KUKA KRL program: FOLLOWTRIG.src, FOLLOWTRIG.dat

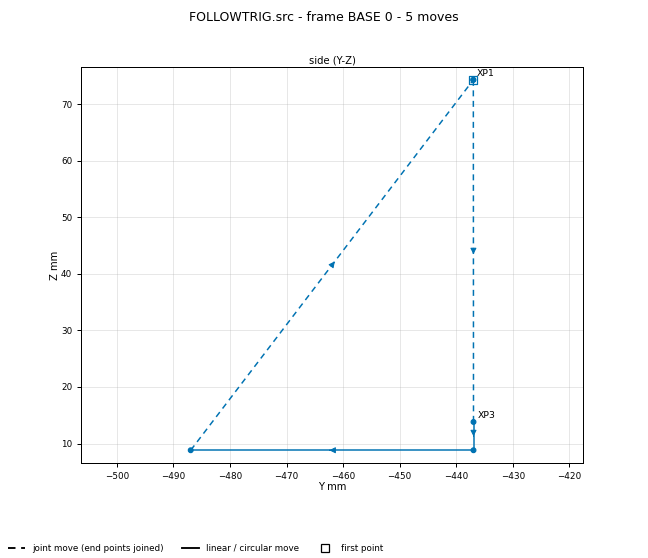
[picture p0: tool path of FOLLOWTRIG.src in frame BASE 0, 5 of 5 moves have a stored position in this frame; points joined in program order, loops and branches not executed]
--- FOLLOWTRIG.src ---
&ACCESS RVO
&REL 127
&PARAM TEMPLATE = C:\KRC\Roboter\Template\vorgabe
&PARAM EDITMASK = *
DEF FOLLOWTRIG( )
DECL TORQUE_TCP_EST MyTorque
DECL BOOL TEMP, HEMP, DEMP
DECL INT TMP1, n, result
DECL INT md_int[16]
DECL REAL md_real[16]
;FOLD INI
  ;FOLD BASISTECH INI
    GLOBAL INTERRUPT DECL 3 WHEN $STOPMESS==TRUE DO IR_STOPM ( )
    INTERRUPT ON 3
    BAS (#INITMOV,0 )
  ;ENDFOLD (BASISTECH INI)
  ;FOLD USER INI
    ;Make your modifications here
  ;ENDFOLD (USER INI)
;ENDFOLD (INI)

$OV_PRO=50
$TOOL=TOOL_DATA[5]
$VEL.CP=1.0
$VEL.ORI1=150
$VEL.ORI2=100
$ACC.CP=1.7
$ACC.ORI1=80
$ACC.ORI2=80
$ORI_TYPE=#CONSTANT

;FOLD PTP P1 Vel=100 % PDAT1 Tool[5]:Pneumatic_gripper_probe Base[0];%{PE}%R 5.6.11,%MKUKATPBASIS,%CMOVE,%VPTP,%P 1:PTP, 2:P1, 3:, 5:100, 7:PDAT1
$BWDSTART=FALSE
PDAT_ACT=PPDAT1
FDAT_ACT=FP1
BAS(#PTP_PARAMS,100)
PTP XP1
;ENDFOLD

;FOLD PTP P3 Vel=100 % PDAT3 Tool[5]:Pneumatic_gripper_probe Base[0];%{PE}%R 5.6.11,%MKUKATPBASIS,%CMOVE,%VPTP,%P 1:PTP, 2:P3, 3:, 5:100, 7:PDAT3
$BWDSTART=FALSE
PDAT_ACT=PPDAT3
FDAT_ACT=FP3
BAS(#PTP_PARAMS,100)
PTP XP3
;ENDFOLD

$STIFFNESS.STRATEGY=10
$STIFFNESS.COMMIT=TRUE
$OV_PRO=25

HALT

HEMP=TRIG()

$OV_PRO=25

LIN_REL {Z -5}

;REPEAT
  ;MyTorque=$TORQUE_TCP_EST
;UNTIL MyTorque.FT.Z >= .1

LIN_REL {Y -50}

HALT

FOR n=1 TO 16
  md_int[n]=0
  md_real[n]=0
ENDFOR

md_real[1]=0.05

result=MD_CMD("PAPAS","TRIGBYCONTACT",md_int[],md_real[])

$STIFFNESS.STRATEGY=10
$STIFFNESS.COMMIT=TRUE
$OV_PRO=25

;FOLD PTP P2 Vel=100 % PDAT2 Tool[5]:Pneumatic_gripper_probe Base[0];%{PE}%R 5.6.11,%MKUKATPBASIS,%CMOVE,%VPTP,%P 1:PTP, 2:P2, 3:, 5:100, 7:PDAT2
$BWDSTART=FALSE
PDAT_ACT=PPDAT2
FDAT_ACT=FP2
BAS(#PTP_PARAMS,100)
PTP XP2
;ENDFOLD

END

--- FOLLOWTRIG.dat ---
&ACCESS RVO
&REL 127
&PARAM TEMPLATE = C:\KRC\Roboter\Template\vorgabe
&PARAM EDITMASK = *
DEFDAT  FOLLOWTRIG
;FOLD EXTERNAL DECLARATIONS;%{PE}%MKUKATPBASIS,%CEXT,%VCOMMON,%P
;FOLD BASISTECH EXT;%{PE}%MKUKATPBASIS,%CEXT,%VEXT,%P
EXT  BAS (BAS_COMMAND  :IN,REAL  :IN )
DECL INT SUCCESS
;ENDFOLD (BASISTECH EXT)
;FOLD USER EXT;%{E}%MKUKATPUSER,%CEXT,%VEXT,%P
;Make here your modifications

;ENDFOLD (USER EXT)
;ENDFOLD (EXTERNAL DECLARATIONS)
DECL BASIS_SUGG_T LAST_BASIS={POINT1[] "P3                      ",POINT2[] "P3                      ",CP_PARAMS[] "CPDAT0                  ",PTP_PARAMS[] "PDAT3                   ",CONT[] "                        ",CP_VEL[] "2.0                     ",PTP_VEL[] "100                     ",SYNC_PARAMS[] "SYNCDAT                 ",SPL_NAME[] "S0                      "}
DECL E6POS XP1={X -559.982727,Y -436.976105,Z 74.2944412,A 89.9887924,B -0.00345713296,C 179.995499,S 1,T 12,E1 0.251655608,E2 0.0,E3 0.0,E4 0.0,E5 0.0,E6 0.0}
DECL FDAT FP1={TOOL_NO 5,BASE_NO 0,IPO_FRAME #BASE,POINT2[] " ",TQ_STATE FALSE}
DECL PDAT PPDAT1={VEL 100.0,ACC 100.0,APO_DIST 100.0,APO_MODE #CPTP}
DECL E6POS XP2={X -559.982422,Y -436.976501,Z 74.2944412,A 89.9887466,B -0.00337572605,C 179.995407,S 1,T 12,E1 0.251655608,E2 0.0,E3 0.0,E4 0.0,E5 0.0,E6 0.0}
DECL FDAT FP2={TOOL_NO 5,BASE_NO 0,IPO_FRAME #BASE,POINT2[] " ",TQ_STATE FALSE}
DECL PDAT PPDAT2={VEL 100.0,ACC 100.0,APO_DIST 100.0,APO_MODE #CPTP}
DECL INT LAST_XP_POINT=2
DECL E6POS XP3={X -559.928772,Y -436.946411,Z 13.8073597,A 89.9849319,B -0.0102660097,C 179.986099,S 1,T 12,E1 0.251947403,E2 0.0,E3 0.0,E4 0.0,E5 0.0,E6 0.0}
DECL FDAT FP3={TOOL_NO 5,BASE_NO 0,IPO_FRAME #BASE,POINT2[] " ",TQ_STATE FALSE}
DECL PDAT PPDAT3={VEL 100.0,ACC 100.0,APO_DIST 100.0,APO_MODE #CPTP}
ENDDAT
